// TIA Portal project "TB_demo2" (V15.1)
// demo de las tablas de observacion

(* hardware
DEVICE "S7-1200 station_1"  S7-1200 Station
   slot 0: "Rack_0"  S7-1200 Rack  Rack  V1.0
   slot 1: "PLC_1"  CPU 1214C AC/DC/Rly  6ES7 214-1BG40-0XB0  V4.2
   slot 3: "AQ 1x12BIT_1"  AQ1 signal board  6ES7 232-4HA30-0XB0  V1.0
*)

// ===== PLC "PLC_1"  CPU 1214C AC/DC/Rly =====

VAR_GLOBAL   // PLC tag table "Tabla de variables estándar"
   "Tag_1" AT %IW64 : Int;
   "Tag_2" AT %MD60 : Real;
   "Tag_3" AT %MD100 : DWord;
   "Tag_4" AT %Q0.0 : Bool;
   "Tag_5" AT %QW80 : Word;
END_VAR

ORGANIZATION_BLOCK "Main"   // OB1, LAD, ProgramCycle
TITLE = "Main Program Sweep (Cycle)"
{ S7_Optimized_Access := 'TRUE' }
VERSION : 0.1
   VAR_INPUT
      Initial_Call : Bool;   // Initial call of this OB
      Remanence : Bool;   // =True, if remanent data are available
   END_VAR
BEGIN

REGION Network 1
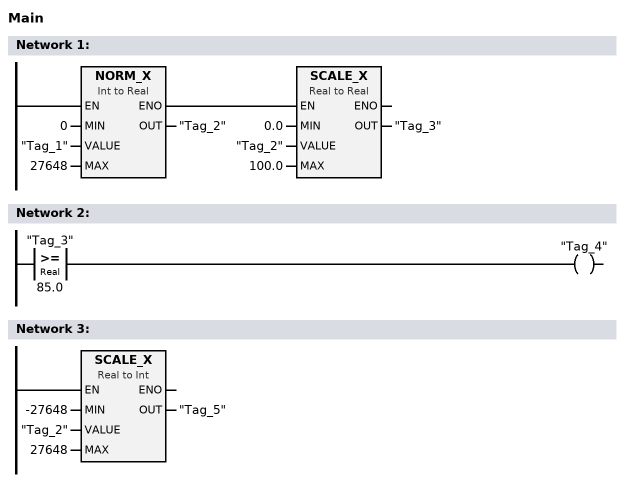
   RUNG wire#powerrail
      { S7_Templates := "[SrcType := Int, DestType := Real]" } Normalize(min := 0, value := "Tag_1", max := 27648, out => "Tag_2")
      { S7_Templates := "[SrcType := Real, DestType := Real]" } Scale(min := 0.0, value := "Tag_2", max := 100.0, out => "Tag_3")
   END_RUNG
   // the same network as SCL:
   "Tag_2" := NORM_X(MIN := 0, VALUE := "Tag_1", MAX := 27648);
   "Tag_3" := SCALE_X(MIN := 0.0, VALUE := "Tag_2", MAX := 100.0);
END_REGION

REGION Network 2
   RUNG wire#powerrail
      { S7_Templates := "SrcType := Real" } GE_Contact(in1 := "Tag_3", in2 := 85.0)
      Coil( "Tag_4" )
   END_RUNG
   // the same network as SCL:
   "Tag_4" := "Tag_3" >= 85.0;
END_REGION

REGION Network 3
   RUNG wire#powerrail
      { S7_Templates := "[SrcType := Real, DestType := Int]" } Scale(min := -27648, value := "Tag_2", max := 27648, out => "Tag_5")
   END_RUNG
   // the same network as SCL:
   "Tag_5" := SCALE_X(MIN := -27648, VALUE := "Tag_2", MAX := 27648);
END_REGION
END_ORGANIZATION_BLOCK